Staubli VAL3: Day21.dtx

num nResult
num nStart[2]
num nEyes
num nDice
num nPointsP1_virt
num nPointsP1_sum
num nPointsP2_virt
num nPointsP2_sum
